TYPE VFD :
STRUCT
	bStart : BOOL;
	bStop : BOOL;
	nRPMSetPointScaled : REAL;
	nRPMFeedBackScaled : REAL;
	nRPMFeedBackRaw : INT;
	
	nRPMSetPointRaw : INT;

	
END_STRUCT
END_TYPE

(* stored: Version 1.1.0.1, ProductVersion 3.1.4024.3
   DUT VFD: Id {4ec55cec-7669-463b-bccf-0e0c2174cc47} *)
